{attribute 'qualified_only'}
VAR_GLOBAL
	
	aCalibPumps         : ARRAY[1..10] OF ST_CalibrationPump;
    bStartCalibration   : BOOL;
    bAbortCalibration   : BOOL;
    bCalibrationRunning : BOOL;
    bCalibrationDone    : BOOL;
    eCalibSolvent       : E_SolventType;
    tDelayStart         : TIME;
    bPrintWhenComplete  : BOOL;
    sGlobalStatus       : STRING[100];
	iPercentLoadBar     : UINT;
	iReplicatesSetpoint : UINT := 1; 
	rAcceptanceCriteria	: LREAL;
	iAllowableFailures	: UINT := 2;
	fbScaleDevice		: FB_ScaleDevice; //Scale Instance Object
	iResultIndex	 	: INT;		 	// Array index on calibration results
	
	aCalibLinearPumps	: ARRAY[1..10] OF ST_LinearPumpCalibration;
	eLeakTestState 		: E_LeakTestState	:= E_LeakTestState.IDLE;
	
	//aCalibCheckResult	: ARRAY[1..100] OF ST_CalibrationPumpResult;
	
	(* Calibration Report*)// -----------------------------------------------------------------------------------------------
	//																													 	|
	stPumpCalReportInfo 	: ST_ReportInfo;	  	//																	  	|
	stPumpCalibrationInfo 	: ST_CalibrationInfo;	//																		|
	stPumpCalibrationData 	: ARRAY[1..100] OF ST_CalibrationData;	//
	//																	
	stLinearCalibrationData : ARRAY[1..10] OF ST_LinearPumpControllDB; // Linear Calibration changing position data from HMI
	//																														|		
	bStartCreationCalJson	: BOOL; // Flag to start the Json creation														|
	bCreationCalJsonDone	: BOOL; // Flag to indicate Json was created Correctly											|
	bCreationCalJsonError	: BOOL; // Flag to indicate Error on Json creation												|
	//																														|
	(**)//-------------------------------------------------------------------------------------------------------------------
	
END_VAR

(* stored: Version 1.1.0.1, ProductVersion 3.1.4024.15
   GVL GVL_Calibration: Id {9a8016f3-cd35-40ee-8da9-49ce7f03d787} *)
